// TIA Portal V19 export
FUNCTION "INPUT" : Void   // FC2, LAD
{ S7_Optimized_Access := 'TRUE' }
// stored: SetENOAutomatically false
BEGIN

REGION Network 1: EMERGENCY_STOP
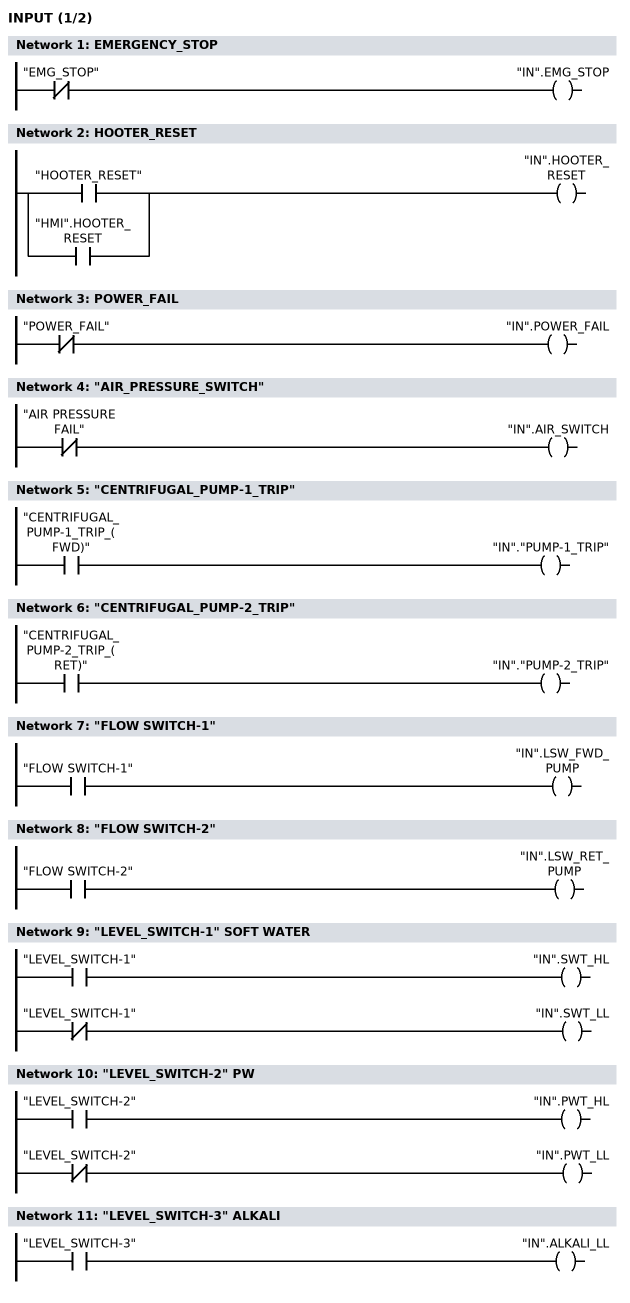
   RUNG wire#powerrail
      I_Contact( "EMG_STOP" )
      Coil( "IN".EMG_STOP )
   END_RUNG
   // the same network as SCL:
   "IN".EMG_STOP := NOT "EMG_STOP";
END_REGION

REGION Network 2: HOOTER_RESET
   RUNG wire#powerrail
      Contact( "HOOTER_RESET" )
      wire#w1
      Coil( "IN".HOOTER_RESET )
   END_RUNG
   RUNG wire#powerrail
      Contact( "HMI".HOOTER_RESET )
   END_RUNG wire#w1
   // the same network as SCL:
   "IN".HOOTER_RESET := "HOOTER_RESET" OR "HMI".HOOTER_RESET;
END_REGION

REGION Network 3: POWER_FAIL
   RUNG wire#powerrail
      I_Contact( "POWER_FAIL" )
      Coil( "IN".POWER_FAIL )
   END_RUNG
   // the same network as SCL:
   "IN".POWER_FAIL := NOT "POWER_FAIL";
END_REGION

REGION Network 4: "AIR_PRESSURE_SWITCH"
   RUNG wire#powerrail
      I_Contact( "AIR PRESSURE FAIL" )
      Coil( "IN".AIR_SWITCH )
   END_RUNG
   // the same network as SCL:
   "IN".AIR_SWITCH := NOT "AIR PRESSURE FAIL";
END_REGION

REGION Network 5: "CENTRIFUGAL_PUMP-1_TRIP"
   RUNG wire#powerrail
      Contact( "CENTRIFUGAL_PUMP-1_TRIP_(FWD)" )
      Coil( "IN"."PUMP-1_TRIP" )
   END_RUNG
   // the same network as SCL:
   "IN"."PUMP-1_TRIP" := "CENTRIFUGAL_PUMP-1_TRIP_(FWD)";
END_REGION

REGION Network 6: "CENTRIFUGAL_PUMP-2_TRIP"
   RUNG wire#powerrail
      Contact( "CENTRIFUGAL_PUMP-2_TRIP_(RET)" )
      Coil( "IN"."PUMP-2_TRIP" )
   END_RUNG
   // the same network as SCL:
   "IN"."PUMP-2_TRIP" := "CENTRIFUGAL_PUMP-2_TRIP_(RET)";
END_REGION

REGION Network 7: "FLOW SWITCH-1"
   RUNG wire#powerrail
      Contact( "FLOW SWITCH-1" )
      Coil( "IN".LSW_FWD_PUMP )
   END_RUNG
   // the same network as SCL:
   "IN".LSW_FWD_PUMP := "FLOW SWITCH-1";
END_REGION

REGION Network 8: "FLOW SWITCH-2"
   RUNG wire#powerrail
      Contact( "FLOW SWITCH-2" )
      Coil( "IN".LSW_RET_PUMP )
   END_RUNG
   // the same network as SCL:
   "IN".LSW_RET_PUMP := "FLOW SWITCH-2";
END_REGION

REGION Network 9: "LEVEL_SWITCH-1" SOFT WATER
   RUNG wire#powerrail
      Contact( "LEVEL_SWITCH-1" )
      Coil( "IN".SWT_HL )
   END_RUNG
   RUNG wire#powerrail
      I_Contact( "LEVEL_SWITCH-1" )
      Coil( "IN".SWT_LL )
   END_RUNG
   // the same network as SCL:
   "IN".SWT_HL := "LEVEL_SWITCH-1";
   "IN".SWT_LL := NOT "LEVEL_SWITCH-1";
END_REGION

REGION Network 10: "LEVEL_SWITCH-2" PW
   RUNG wire#powerrail
      Contact( "LEVEL_SWITCH-2" )
      Coil( "IN".PWT_HL )
   END_RUNG
   RUNG wire#powerrail
      I_Contact( "LEVEL_SWITCH-2" )
      Coil( "IN".PWT_LL )
   END_RUNG
   // the same network as SCL:
   "IN".PWT_HL := "LEVEL_SWITCH-2";
   "IN".PWT_LL := NOT "LEVEL_SWITCH-2";
END_REGION

REGION Network 11: "LEVEL_SWITCH-3" ALKALI
   RUNG wire#powerrail
      Contact( "LEVEL_SWITCH-3" )
      Coil( "IN".ALKALI_LL )
   END_RUNG
   // the same network as SCL:
   "IN".ALKALI_LL := "LEVEL_SWITCH-3";
END_REGION

REGION Network 12: "LEVEL_SWITCH-4"ACID
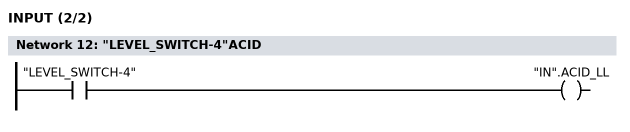
   RUNG wire#powerrail
      Contact( "LEVEL_SWITCH-4" )
      Coil( "IN".ACID_LL )
   END_RUNG
   // the same network as SCL:
   "IN".ACID_LL := "LEVEL_SWITCH-4";
END_REGION
END_FUNCTION
